// TIA Portal V19 export
FUNCTION "Digital_IN" : Void   // FC1, LAD
{ S7_Optimized_Access := 'TRUE' }
// stored: SetENOAutomatically false
BEGIN

REGION Network 1: Safety OK
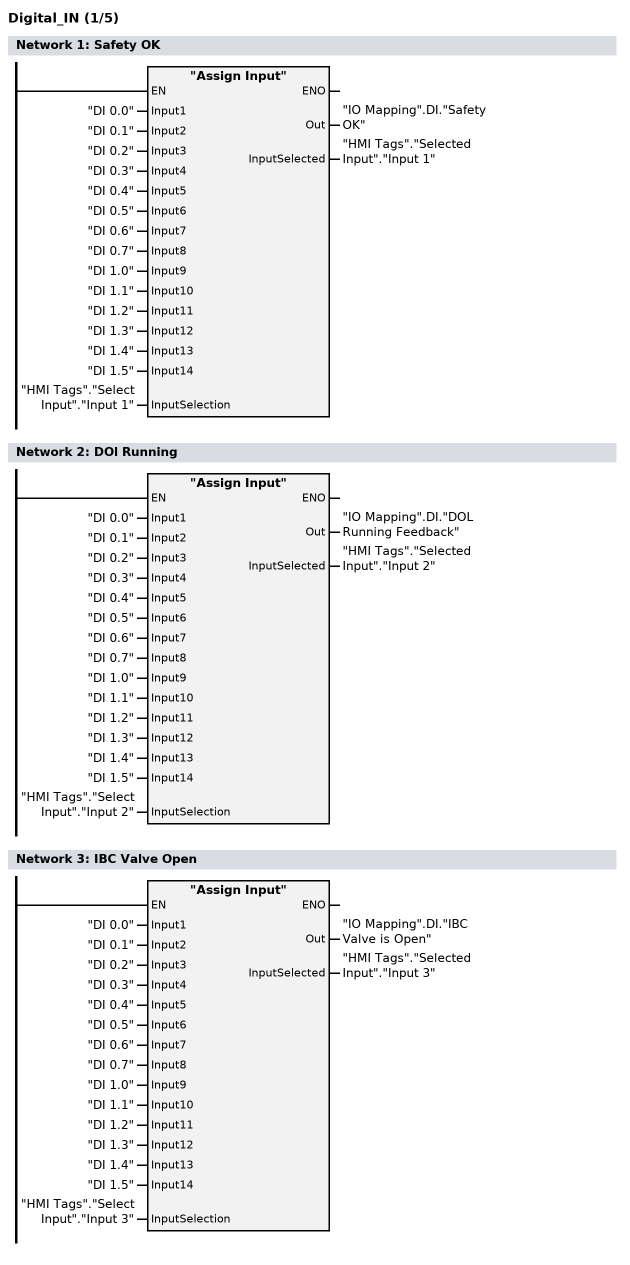
   RUNG wire#powerrail
      "Assign Input"(Input1 := "DI 0.0", Input2 := "DI 0.1", Input3 := "DI 0.2", Input4 := "DI 0.3", Input5 := "DI 0.4", Input6 := "DI 0.5", Input7 := "DI 0.6", Input8 := "DI 0.7", Input9 := "DI 1.0", Input10 := "DI 1.1", Input11 := "DI 1.2", Input12 := "DI 1.3", Input13 := "DI 1.4", Input14 := "DI 1.5", InputSelection := "HMI Tags"."Select Input"."Input 1", Out => "IO Mapping".DI."Safety OK", InputSelected => "HMI Tags"."Selected Input"."Input 1")
   END_RUNG
   // the same network as SCL:
   "Assign Input"(Input1 := "DI 0.0",
                  Input2 := "DI 0.1",
                  Input3 := "DI 0.2",
                  Input4 := "DI 0.3",
                  Input5 := "DI 0.4",
                  Input6 := "DI 0.5",
                  Input7 := "DI 0.6",
                  Input8 := "DI 0.7",
                  Input9 := "DI 1.0",
                  Input10 := "DI 1.1",
                  Input11 := "DI 1.2",
                  Input12 := "DI 1.3",
                  Input13 := "DI 1.4",
                  Input14 := "DI 1.5",
                  InputSelection := "HMI Tags"."Select Input"."Input 1",
                  Out => "IO Mapping".DI."Safety OK",
                  InputSelected => "HMI Tags"."Selected Input"."Input 1");
END_REGION

REGION Network 2: DOl Running
   RUNG wire#powerrail
      "Assign Input"(Input1 := "DI 0.0", Input2 := "DI 0.1", Input3 := "DI 0.2", Input4 := "DI 0.3", Input5 := "DI 0.4", Input6 := "DI 0.5", Input7 := "DI 0.6", Input8 := "DI 0.7", Input9 := "DI 1.0", Input10 := "DI 1.1", Input11 := "DI 1.2", Input12 := "DI 1.3", Input13 := "DI 1.4", Input14 := "DI 1.5", InputSelection := "HMI Tags"."Select Input"."Input 2", Out => "IO Mapping".DI."DOL Running Feedback", InputSelected => "HMI Tags"."Selected Input"."Input 2")
   END_RUNG
   // the same network as SCL:
   "Assign Input"(Input1 := "DI 0.0",
                  Input2 := "DI 0.1",
                  Input3 := "DI 0.2",
                  Input4 := "DI 0.3",
                  Input5 := "DI 0.4",
                  Input6 := "DI 0.5",
                  Input7 := "DI 0.6",
                  Input8 := "DI 0.7",
                  Input9 := "DI 1.0",
                  Input10 := "DI 1.1",
                  Input11 := "DI 1.2",
                  Input12 := "DI 1.3",
                  Input13 := "DI 1.4",
                  Input14 := "DI 1.5",
                  InputSelection := "HMI Tags"."Select Input"."Input 2",
                  Out => "IO Mapping".DI."DOL Running Feedback",
                  InputSelected => "HMI Tags"."Selected Input"."Input 2");
END_REGION

REGION Network 3: IBC Valve Open
   RUNG wire#powerrail
      "Assign Input"(Input1 := "DI 0.0", Input2 := "DI 0.1", Input3 := "DI 0.2", Input4 := "DI 0.3", Input5 := "DI 0.4", Input6 := "DI 0.5", Input7 := "DI 0.6", Input8 := "DI 0.7", Input9 := "DI 1.0", Input10 := "DI 1.1", Input11 := "DI 1.2", Input12 := "DI 1.3", Input13 := "DI 1.4", Input14 := "DI 1.5", InputSelection := "HMI Tags"."Select Input"."Input 3", Out => "IO Mapping".DI."IBC Valve is Open", InputSelected => "HMI Tags"."Selected Input"."Input 3")
   END_RUNG
   // the same network as SCL:
   "Assign Input"(Input1 := "DI 0.0",
                  Input2 := "DI 0.1",
                  Input3 := "DI 0.2",
                  Input4 := "DI 0.3",
                  Input5 := "DI 0.4",
                  Input6 := "DI 0.5",
                  Input7 := "DI 0.6",
                  Input8 := "DI 0.7",
                  Input9 := "DI 1.0",
                  Input10 := "DI 1.1",
                  Input11 := "DI 1.2",
                  Input12 := "DI 1.3",
                  Input13 := "DI 1.4",
                  Input14 := "DI 1.5",
                  InputSelection := "HMI Tags"."Select Input"."Input 3",
                  Out => "IO Mapping".DI."IBC Valve is Open",
                  InputSelected => "HMI Tags"."Selected Input"."Input 3");
END_REGION

REGION Network 4: IBC Valve closed
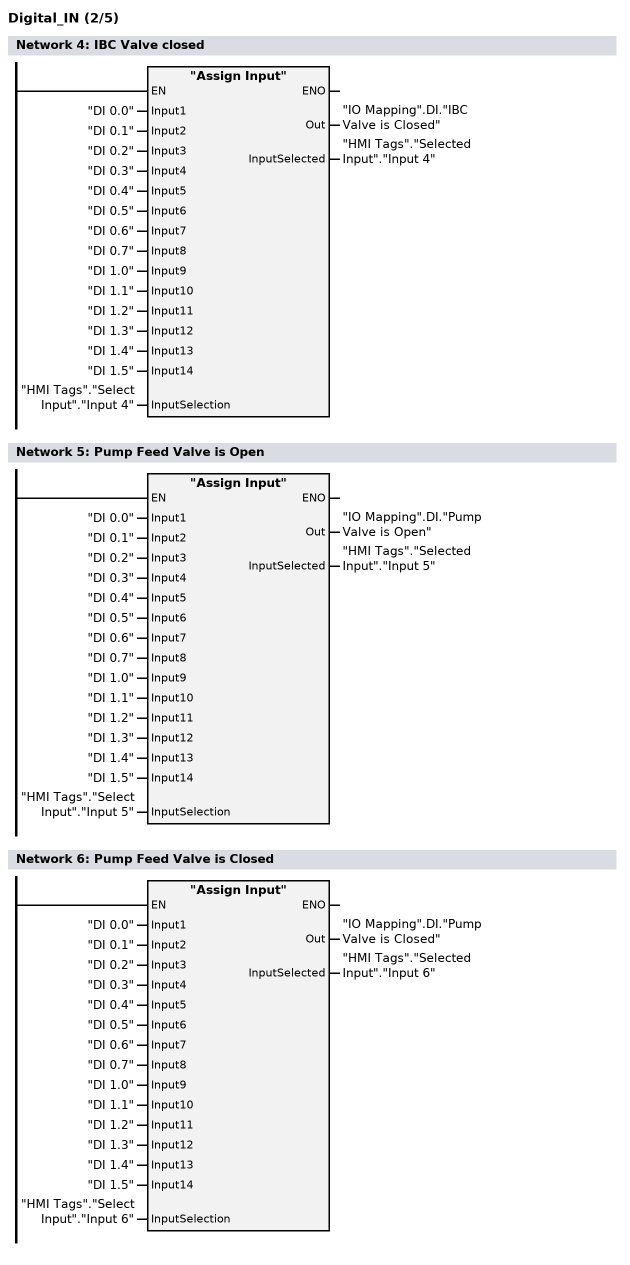
   RUNG wire#powerrail
      "Assign Input"(Input1 := "DI 0.0", Input2 := "DI 0.1", Input3 := "DI 0.2", Input4 := "DI 0.3", Input5 := "DI 0.4", Input6 := "DI 0.5", Input7 := "DI 0.6", Input8 := "DI 0.7", Input9 := "DI 1.0", Input10 := "DI 1.1", Input11 := "DI 1.2", Input12 := "DI 1.3", Input13 := "DI 1.4", Input14 := "DI 1.5", InputSelection := "HMI Tags"."Select Input"."Input 4", Out => "IO Mapping".DI."IBC Valve is Closed", InputSelected => "HMI Tags"."Selected Input"."Input 4")
   END_RUNG
   // the same network as SCL:
   "Assign Input"(Input1 := "DI 0.0",
                  Input2 := "DI 0.1",
                  Input3 := "DI 0.2",
                  Input4 := "DI 0.3",
                  Input5 := "DI 0.4",
                  Input6 := "DI 0.5",
                  Input7 := "DI 0.6",
                  Input8 := "DI 0.7",
                  Input9 := "DI 1.0",
                  Input10 := "DI 1.1",
                  Input11 := "DI 1.2",
                  Input12 := "DI 1.3",
                  Input13 := "DI 1.4",
                  Input14 := "DI 1.5",
                  InputSelection := "HMI Tags"."Select Input"."Input 4",
                  Out => "IO Mapping".DI."IBC Valve is Closed",
                  InputSelected => "HMI Tags"."Selected Input"."Input 4");
END_REGION

REGION Network 5: Pump Feed Valve is Open
   RUNG wire#powerrail
      "Assign Input"(Input1 := "DI 0.0", Input2 := "DI 0.1", Input3 := "DI 0.2", Input4 := "DI 0.3", Input5 := "DI 0.4", Input6 := "DI 0.5", Input7 := "DI 0.6", Input8 := "DI 0.7", Input9 := "DI 1.0", Input10 := "DI 1.1", Input11 := "DI 1.2", Input12 := "DI 1.3", Input13 := "DI 1.4", Input14 := "DI 1.5", InputSelection := "HMI Tags"."Select Input"."Input 5", Out => "IO Mapping".DI."Pump Valve is Open", InputSelected => "HMI Tags"."Selected Input"."Input 5")
   END_RUNG
   // the same network as SCL:
   "Assign Input"(Input1 := "DI 0.0",
                  Input2 := "DI 0.1",
                  Input3 := "DI 0.2",
                  Input4 := "DI 0.3",
                  Input5 := "DI 0.4",
                  Input6 := "DI 0.5",
                  Input7 := "DI 0.6",
                  Input8 := "DI 0.7",
                  Input9 := "DI 1.0",
                  Input10 := "DI 1.1",
                  Input11 := "DI 1.2",
                  Input12 := "DI 1.3",
                  Input13 := "DI 1.4",
                  Input14 := "DI 1.5",
                  InputSelection := "HMI Tags"."Select Input"."Input 5",
                  Out => "IO Mapping".DI."Pump Valve is Open",
                  InputSelected => "HMI Tags"."Selected Input"."Input 5");
END_REGION

REGION Network 6: Pump Feed Valve is Closed
   RUNG wire#powerrail
      "Assign Input"(Input1 := "DI 0.0", Input2 := "DI 0.1", Input3 := "DI 0.2", Input4 := "DI 0.3", Input5 := "DI 0.4", Input6 := "DI 0.5", Input7 := "DI 0.6", Input8 := "DI 0.7", Input9 := "DI 1.0", Input10 := "DI 1.1", Input11 := "DI 1.2", Input12 := "DI 1.3", Input13 := "DI 1.4", Input14 := "DI 1.5", InputSelection := "HMI Tags"."Select Input"."Input 6", Out => "IO Mapping".DI."Pump Valve is Closed", InputSelected => "HMI Tags"."Selected Input"."Input 6")
   END_RUNG
   // the same network as SCL:
   "Assign Input"(Input1 := "DI 0.0",
                  Input2 := "DI 0.1",
                  Input3 := "DI 0.2",
                  Input4 := "DI 0.3",
                  Input5 := "DI 0.4",
                  Input6 := "DI 0.5",
                  Input7 := "DI 0.6",
                  Input8 := "DI 0.7",
                  Input9 := "DI 1.0",
                  Input10 := "DI 1.1",
                  Input11 := "DI 1.2",
                  Input12 := "DI 1.3",
                  Input13 := "DI 1.4",
                  Input14 := "DI 1.5",
                  InputSelection := "HMI Tags"."Select Input"."Input 6",
                  Out => "IO Mapping".DI."Pump Valve is Closed",
                  InputSelected => "HMI Tags"."Selected Input"."Input 6");
END_REGION

REGION Network 7: Flometer Feed Valve is Open
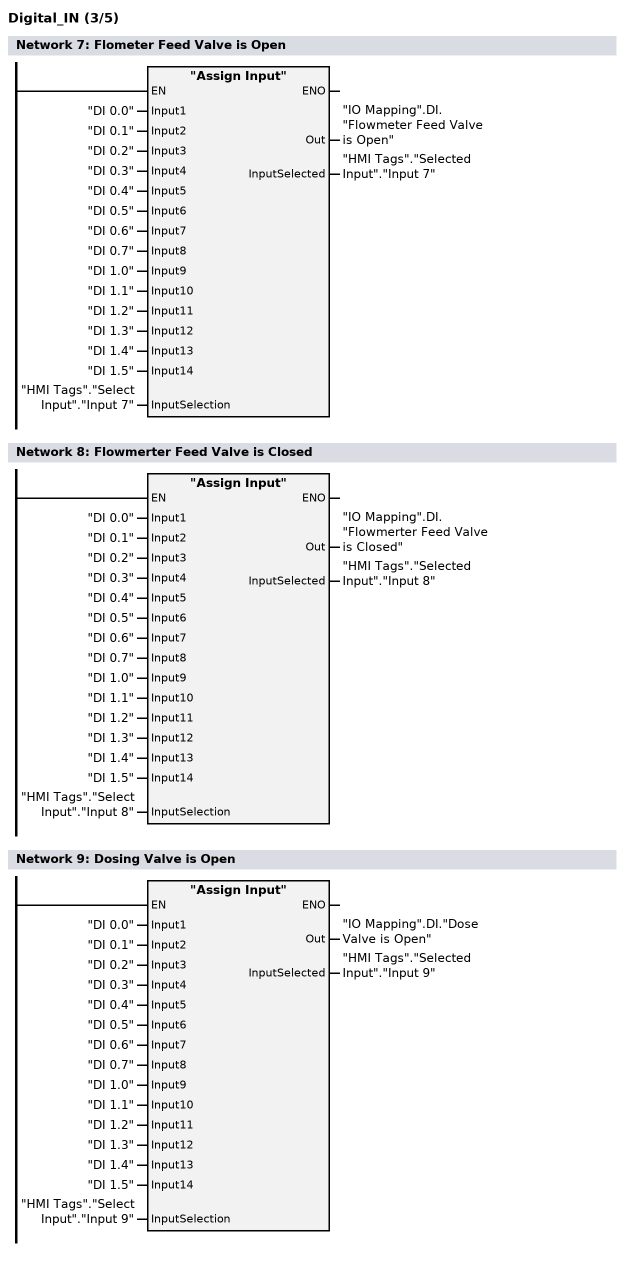
   RUNG wire#powerrail
      "Assign Input"(Input1 := "DI 0.0", Input2 := "DI 0.1", Input3 := "DI 0.2", Input4 := "DI 0.3", Input5 := "DI 0.4", Input6 := "DI 0.5", Input7 := "DI 0.6", Input8 := "DI 0.7", Input9 := "DI 1.0", Input10 := "DI 1.1", Input11 := "DI 1.2", Input12 := "DI 1.3", Input13 := "DI 1.4", Input14 := "DI 1.5", InputSelection := "HMI Tags"."Select Input"."Input 7", Out => "IO Mapping".DI."Flowmeter Feed Valve is Open", InputSelected => "HMI Tags"."Selected Input"."Input 7")
   END_RUNG
   // the same network as SCL:
   "Assign Input"(Input1 := "DI 0.0",
                  Input2 := "DI 0.1",
                  Input3 := "DI 0.2",
                  Input4 := "DI 0.3",
                  Input5 := "DI 0.4",
                  Input6 := "DI 0.5",
                  Input7 := "DI 0.6",
                  Input8 := "DI 0.7",
                  Input9 := "DI 1.0",
                  Input10 := "DI 1.1",
                  Input11 := "DI 1.2",
                  Input12 := "DI 1.3",
                  Input13 := "DI 1.4",
                  Input14 := "DI 1.5",
                  InputSelection := "HMI Tags"."Select Input"."Input 7",
                  Out => "IO Mapping".DI."Flowmeter Feed Valve is Open",
                  InputSelected => "HMI Tags"."Selected Input"."Input 7");
END_REGION

REGION Network 8: Flowmerter Feed Valve is Closed
   RUNG wire#powerrail
      "Assign Input"(Input1 := "DI 0.0", Input2 := "DI 0.1", Input3 := "DI 0.2", Input4 := "DI 0.3", Input5 := "DI 0.4", Input6 := "DI 0.5", Input7 := "DI 0.6", Input8 := "DI 0.7", Input9 := "DI 1.0", Input10 := "DI 1.1", Input11 := "DI 1.2", Input12 := "DI 1.3", Input13 := "DI 1.4", Input14 := "DI 1.5", InputSelection := "HMI Tags"."Select Input"."Input 8", Out => "IO Mapping".DI."Flowmerter Feed Valve is Closed", InputSelected => "HMI Tags"."Selected Input"."Input 8")
   END_RUNG
   // the same network as SCL:
   "Assign Input"(Input1 := "DI 0.0",
                  Input2 := "DI 0.1",
                  Input3 := "DI 0.2",
                  Input4 := "DI 0.3",
                  Input5 := "DI 0.4",
                  Input6 := "DI 0.5",
                  Input7 := "DI 0.6",
                  Input8 := "DI 0.7",
                  Input9 := "DI 1.0",
                  Input10 := "DI 1.1",
                  Input11 := "DI 1.2",
                  Input12 := "DI 1.3",
                  Input13 := "DI 1.4",
                  Input14 := "DI 1.5",
                  InputSelection := "HMI Tags"."Select Input"."Input 8",
                  Out => "IO Mapping".DI."Flowmerter Feed Valve is Closed",
                  InputSelected => "HMI Tags"."Selected Input"."Input 8");
END_REGION

REGION Network 9: Dosing Valve is Open
   RUNG wire#powerrail
      "Assign Input"(Input1 := "DI 0.0", Input2 := "DI 0.1", Input3 := "DI 0.2", Input4 := "DI 0.3", Input5 := "DI 0.4", Input6 := "DI 0.5", Input7 := "DI 0.6", Input8 := "DI 0.7", Input9 := "DI 1.0", Input10 := "DI 1.1", Input11 := "DI 1.2", Input12 := "DI 1.3", Input13 := "DI 1.4", Input14 := "DI 1.5", InputSelection := "HMI Tags"."Select Input"."Input 9", Out => "IO Mapping".DI."Dose Valve is Open", InputSelected => "HMI Tags"."Selected Input"."Input 9")
   END_RUNG
   // the same network as SCL:
   "Assign Input"(Input1 := "DI 0.0",
                  Input2 := "DI 0.1",
                  Input3 := "DI 0.2",
                  Input4 := "DI 0.3",
                  Input5 := "DI 0.4",
                  Input6 := "DI 0.5",
                  Input7 := "DI 0.6",
                  Input8 := "DI 0.7",
                  Input9 := "DI 1.0",
                  Input10 := "DI 1.1",
                  Input11 := "DI 1.2",
                  Input12 := "DI 1.3",
                  Input13 := "DI 1.4",
                  Input14 := "DI 1.5",
                  InputSelection := "HMI Tags"."Select Input"."Input 9",
                  Out => "IO Mapping".DI."Dose Valve is Open",
                  InputSelected => "HMI Tags"."Selected Input"."Input 9");
END_REGION

REGION Network 10: Dosing Valve is Closed
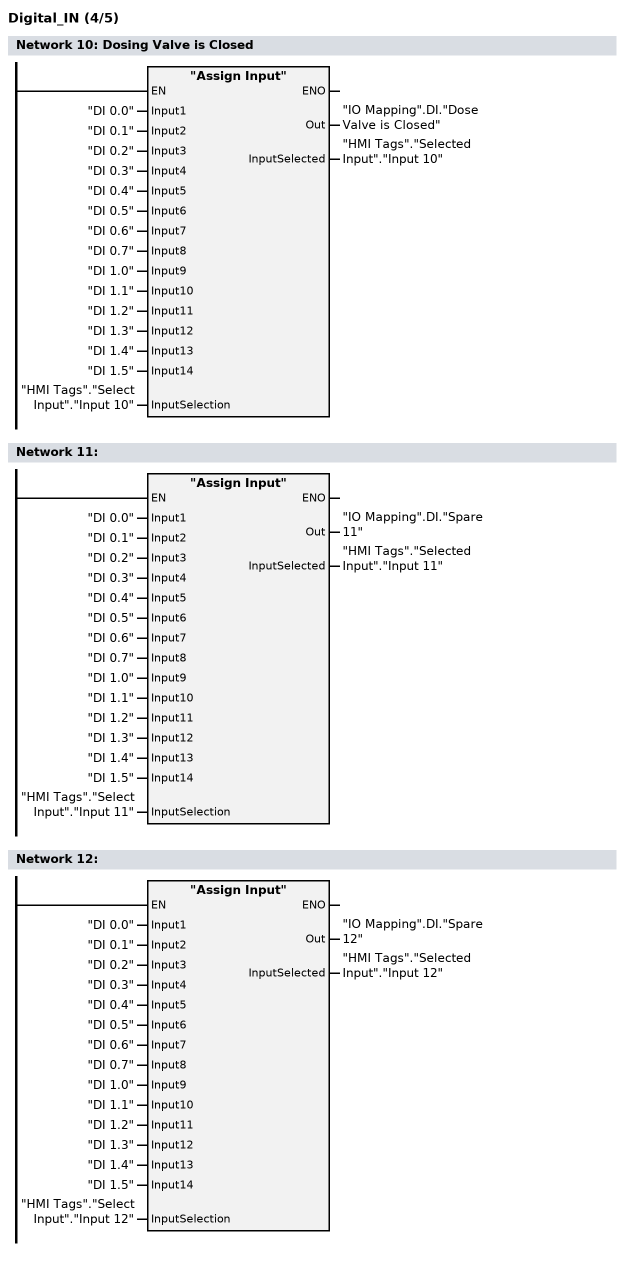
   RUNG wire#powerrail
      "Assign Input"(Input1 := "DI 0.0", Input2 := "DI 0.1", Input3 := "DI 0.2", Input4 := "DI 0.3", Input5 := "DI 0.4", Input6 := "DI 0.5", Input7 := "DI 0.6", Input8 := "DI 0.7", Input9 := "DI 1.0", Input10 := "DI 1.1", Input11 := "DI 1.2", Input12 := "DI 1.3", Input13 := "DI 1.4", Input14 := "DI 1.5", InputSelection := "HMI Tags"."Select Input"."Input 10", Out => "IO Mapping".DI."Dose Valve is Closed", InputSelected => "HMI Tags"."Selected Input"."Input 10")
   END_RUNG
   // the same network as SCL:
   "Assign Input"(Input1 := "DI 0.0",
                  Input2 := "DI 0.1",
                  Input3 := "DI 0.2",
                  Input4 := "DI 0.3",
                  Input5 := "DI 0.4",
                  Input6 := "DI 0.5",
                  Input7 := "DI 0.6",
                  Input8 := "DI 0.7",
                  Input9 := "DI 1.0",
                  Input10 := "DI 1.1",
                  Input11 := "DI 1.2",
                  Input12 := "DI 1.3",
                  Input13 := "DI 1.4",
                  Input14 := "DI 1.5",
                  InputSelection := "HMI Tags"."Select Input"."Input 10",
                  Out => "IO Mapping".DI."Dose Valve is Closed",
                  InputSelected => "HMI Tags"."Selected Input"."Input 10");
END_REGION

REGION Network 11
   RUNG wire#powerrail
      "Assign Input"(Input1 := "DI 0.0", Input2 := "DI 0.1", Input3 := "DI 0.2", Input4 := "DI 0.3", Input5 := "DI 0.4", Input6 := "DI 0.5", Input7 := "DI 0.6", Input8 := "DI 0.7", Input9 := "DI 1.0", Input10 := "DI 1.1", Input11 := "DI 1.2", Input12 := "DI 1.3", Input13 := "DI 1.4", Input14 := "DI 1.5", InputSelection := "HMI Tags"."Select Input"."Input 11", Out => "IO Mapping".DI."Spare 11", InputSelected => "HMI Tags"."Selected Input"."Input 11")
   END_RUNG
   // the same network as SCL:
   "Assign Input"(Input1 := "DI 0.0",
                  Input2 := "DI 0.1",
                  Input3 := "DI 0.2",
                  Input4 := "DI 0.3",
                  Input5 := "DI 0.4",
                  Input6 := "DI 0.5",
                  Input7 := "DI 0.6",
                  Input8 := "DI 0.7",
                  Input9 := "DI 1.0",
                  Input10 := "DI 1.1",
                  Input11 := "DI 1.2",
                  Input12 := "DI 1.3",
                  Input13 := "DI 1.4",
                  Input14 := "DI 1.5",
                  InputSelection := "HMI Tags"."Select Input"."Input 11",
                  Out => "IO Mapping".DI."Spare 11",
                  InputSelected => "HMI Tags"."Selected Input"."Input 11");
END_REGION

REGION Network 12
   RUNG wire#powerrail
      "Assign Input"(Input1 := "DI 0.0", Input2 := "DI 0.1", Input3 := "DI 0.2", Input4 := "DI 0.3", Input5 := "DI 0.4", Input6 := "DI 0.5", Input7 := "DI 0.6", Input8 := "DI 0.7", Input9 := "DI 1.0", Input10 := "DI 1.1", Input11 := "DI 1.2", Input12 := "DI 1.3", Input13 := "DI 1.4", Input14 := "DI 1.5", InputSelection := "HMI Tags"."Select Input"."Input 12", Out => "IO Mapping".DI."Spare 12", InputSelected => "HMI Tags"."Selected Input"."Input 12")
   END_RUNG
   // the same network as SCL:
   "Assign Input"(Input1 := "DI 0.0",
                  Input2 := "DI 0.1",
                  Input3 := "DI 0.2",
                  Input4 := "DI 0.3",
                  Input5 := "DI 0.4",
                  Input6 := "DI 0.5",
                  Input7 := "DI 0.6",
                  Input8 := "DI 0.7",
                  Input9 := "DI 1.0",
                  Input10 := "DI 1.1",
                  Input11 := "DI 1.2",
                  Input12 := "DI 1.3",
                  Input13 := "DI 1.4",
                  Input14 := "DI 1.5",
                  InputSelection := "HMI Tags"."Select Input"."Input 12",
                  Out => "IO Mapping".DI."Spare 12",
                  InputSelected => "HMI Tags"."Selected Input"."Input 12");
END_REGION

REGION Network 13
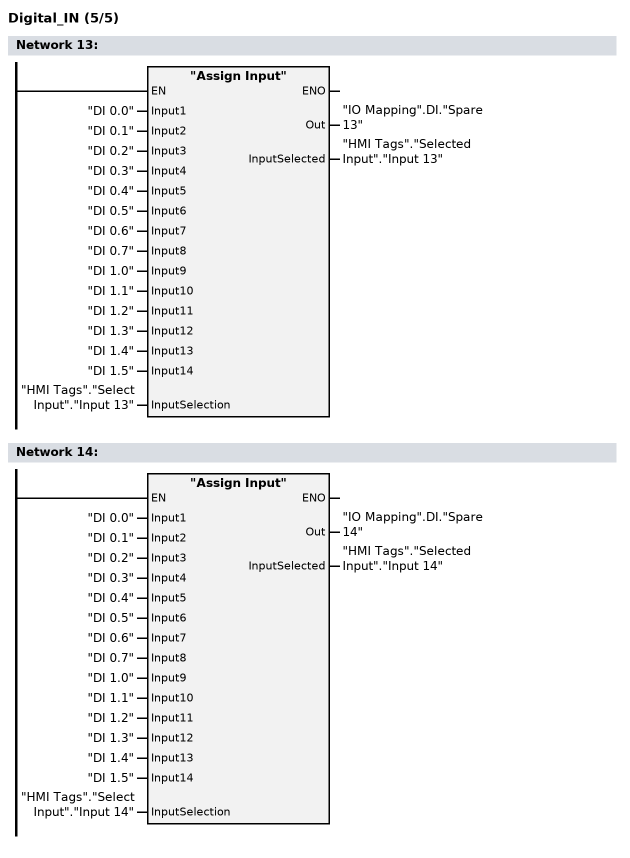
   RUNG wire#powerrail
      "Assign Input"(Input1 := "DI 0.0", Input2 := "DI 0.1", Input3 := "DI 0.2", Input4 := "DI 0.3", Input5 := "DI 0.4", Input6 := "DI 0.5", Input7 := "DI 0.6", Input8 := "DI 0.7", Input9 := "DI 1.0", Input10 := "DI 1.1", Input11 := "DI 1.2", Input12 := "DI 1.3", Input13 := "DI 1.4", Input14 := "DI 1.5", InputSelection := "HMI Tags"."Select Input"."Input 13", Out => "IO Mapping".DI."Spare 13", InputSelected => "HMI Tags"."Selected Input"."Input 13")
   END_RUNG
   // the same network as SCL:
   "Assign Input"(Input1 := "DI 0.0",
                  Input2 := "DI 0.1",
                  Input3 := "DI 0.2",
                  Input4 := "DI 0.3",
                  Input5 := "DI 0.4",
                  Input6 := "DI 0.5",
                  Input7 := "DI 0.6",
                  Input8 := "DI 0.7",
                  Input9 := "DI 1.0",
                  Input10 := "DI 1.1",
                  Input11 := "DI 1.2",
                  Input12 := "DI 1.3",
                  Input13 := "DI 1.4",
                  Input14 := "DI 1.5",
                  InputSelection := "HMI Tags"."Select Input"."Input 13",
                  Out => "IO Mapping".DI."Spare 13",
                  InputSelected => "HMI Tags"."Selected Input"."Input 13");
END_REGION

REGION Network 14
   RUNG wire#powerrail
      "Assign Input"(Input1 := "DI 0.0", Input2 := "DI 0.1", Input3 := "DI 0.2", Input4 := "DI 0.3", Input5 := "DI 0.4", Input6 := "DI 0.5", Input7 := "DI 0.6", Input8 := "DI 0.7", Input9 := "DI 1.0", Input10 := "DI 1.1", Input11 := "DI 1.2", Input12 := "DI 1.3", Input13 := "DI 1.4", Input14 := "DI 1.5", InputSelection := "HMI Tags"."Select Input"."Input 14", Out => "IO Mapping".DI."Spare 14", InputSelected => "HMI Tags"."Selected Input"."Input 14")
   END_RUNG
   // the same network as SCL:
   "Assign Input"(Input1 := "DI 0.0",
                  Input2 := "DI 0.1",
                  Input3 := "DI 0.2",
                  Input4 := "DI 0.3",
                  Input5 := "DI 0.4",
                  Input6 := "DI 0.5",
                  Input7 := "DI 0.6",
                  Input8 := "DI 0.7",
                  Input9 := "DI 1.0",
                  Input10 := "DI 1.1",
                  Input11 := "DI 1.2",
                  Input12 := "DI 1.3",
                  Input13 := "DI 1.4",
                  Input14 := "DI 1.5",
                  InputSelection := "HMI Tags"."Select Input"."Input 14",
                  Out => "IO Mapping".DI."Spare 14",
                  InputSelected => "HMI Tags"."Selected Input"."Input 14");
END_REGION
END_FUNCTION
